(* IEC 61131-3 sources: AutomationLab/, 3 files *)

(* ---- GVL.st ---- *)
// ============================================
// ГЛОБАЛЬНЫЕ ПЕРЕМЕННЫЕ
// ============================================
VAR_GLOBAL
    // Датчик в начале конвейера
    DI_SensorA: BOOL;
    // Датчик в конце конвейера
    DI_SensorB: BOOL;
    // Команда на работу двигателя конвейера
    DO_ComMotor: BOOL;
    // Лампочка на панели оператора: лента работает
    DO_LampRun: BOOL;
END_VAR

(* ---- Readme.st ---- *)
FUNCTION Readme : BOOL
VAR_INPUT
END_VAR
VAR
END_VAR

(*
# Задание: Управление конвейером

## Цель
Учебная задача управления конвейером

## Описание системы
Конвейер перемещает на своей ленте груз. Груз доезжает до датчика на конце ленты и должен там останавиться.

1. Лента вращается.
2. Как только поступит сигнал с оптического НЗ датчика - лента должна прекратить вращение.

## Требования к программе на ПЛК

### 1. Выходы на двигатель конвейера
Выходы ПЛК на двигатель конвейера постоянно включен, пока не сработает НЗ датчик на конце ленты.

## Требования к интерфейсу оператора (ЧМИ)

1. Индикация работы двигателя конвейера одной лампочкой.
2. Лампы индикации сбоев, запретов, ошибок — красные.

## Входы/Выходы (предварительный перечень)

### Входы:
| Имя | Описание | Тип |
|-----|----------|-----|
| SENSOR_A | Датчик на конце ленты | Дискретный |

### Выходы:
| Имя | Описание | Тип |
|-----|----------|-----|
| OUT_MOTOR | Включить двигатель конвейера | Дискретный |

### Требования к оборудованию:
1.  ПЛК – Овен ПЛК210.

## Примечания
- Код писать на ST (Structured Text) с использованием CoDeSys v3.
 *)

(* ---- PLC_PRG.st ---- *)
PROGRAM PLC_PRG
VAR
END_VAR

// ============================================
// ГЛАВНАЯ ЦИКЛИЧНО ВЫЗЫВАЕМАЯ ПРОГРАММА
// ============================================
